// Alarm keypad FB (B11-11-11L11-11-11)
FUNCTION_BLOCK FB_AlarmKeypad IMPLEMENTS I_AlarmKeypad
VAR
	sName			: STRING;				// Keypad name

	fbButton1		: FB_DigitalIn;			// Button 1
	fbLed1			: FB_DigitalOut;		// LED 1
	fbButton2		: FB_DigitalIn;			// Button 2
	fbLed2			: FB_DigitalOut;		// LED 2
	fbButton3		: FB_DigitalIn;			// Button 3
	fbLed3			: FB_DigitalOut;		// LED 3
	fbButton4		: FB_DigitalIn;			// Button 4
	fbLed4			: FB_DigitalOut;		// LED 4
	fbButton5		: FB_DigitalIn;			// Button 5
	fbLed5			: FB_DigitalOut;		// LED 5
	fbButton6		: FB_DigitalIn;			// Button 6
	fbLed6			: FB_DigitalOut;		// LED 6
	fbBuzzer		: FB_DigitalOut;		// Buzzer

	eState			: E_KeypadState;		// Keypad state
	sConfiguredCode	: STRING;				// Configured alarm code
	sInputCode		: STRING;				// User input code
	dtInputTime		: DATE_AND_TIME;		// Date and time of last user input
	stLedsDefault	: ST_LedState;			// Default LEDs state
	
	stHMI			: ST_AlarmKeypadHMI;	// HMI data
	stVirtual		: ST_AlarmKeypadVirtual;	// Virtual keypad
END_VAR

// Returns true if the user input code equals the configured code
METHOD CheckCode : BOOL
// Compare codes
CheckCode := sInputCode = sConfiguredCode;

// Reset input if correct code was entered
IF CheckCode THEN
	Reset();
END_IF
END_METHOD

// Collect user input from buttons and build the entered code, returns true if input was detected
METHOD PRIVATE CollectInput: BOOL
VAR
	sInput			: STRING;
END_VAR
// Check buttons and translate to input
IF fbButton1.Command = E_DICommand.ShortPress THEN sInput := '1'; END_IF
IF fbButton2.Command = E_DICommand.ShortPress THEN sInput := '2'; END_IF
IF fbButton3.Command = E_DICommand.ShortPress THEN sInput := '3'; END_IF
IF fbButton4.Command = E_DICommand.ShortPress THEN sInput := '4'; END_IF
IF fbButton5.Command = E_DICommand.ShortPress THEN sInput := '5'; END_IF
IF fbButton6.Command = E_DICommand.ShortPress THEN sInput := '6'; END_IF

// Check if input was detected
IF sInput <> '' THEN
	// Build user input code
	sInputCode := CONCAT(sInputCode, sInput);
	
	// Update time of last input
	dtInputTime := GetDateTime();
	
	// Set output
	CollectInput := TRUE;
ELSE
	// Set output
	CollectInput := FALSE;
END_IF
END_METHOD

// Run this method every cycle
METHOD Execute
VAR CONSTANT
	stLedsOn	: ST_LedState := (eLed1 := E_DOCommand.On,
									eLed2 := E_DOCommand.On,
									eLed3 := E_DOCommand.On,
									eLed4 := E_DOCommand.On,
									eLed5 := E_DOCommand.On,
									eLed6 := E_DOCommand.On);
END_VAR
// Keypad state machine
CASE eState OF
	E_KeypadState.Init:
		// Initialize
		eState := E_KeypadState.Idle;
	
	E_KeypadState.Idle:
		// Wait for input
		IF CollectInput() THEN
			eState := E_KeypadState.InputDetected;
		END_IF
	
	E_KeypadState.InputDetected:
		// Collect input in every state so no input is lost
		CollectInput();
		
		// Enable all LEDs
		SetLeds(stLedsOn);
		
		eState := E_KeypadState.CheckInput;
		
	E_KeypadState.CheckInput:
		// Continue collecting input
		CollectInput();
		
		// If no input is detected during some time, reset the keypad
		IF GetDateTime() - dtInputTime > T#2S THEN
			eState := E_KeypadState.Reset;
		END_IF
		
	E_KeypadState.Reset:
		// Reset keypad
		Reset();
		
		eState := E_KeypadState.Idle;
END_CASE

// Update HMI
UpdateHMI();
END_METHOD

METHOD FB_init : BOOL
VAR_INPUT
	bInitRetains	: BOOL;		// if TRUE, the retain variables are initialized (warm start / cold start)
	bInCopyCode		: BOOL;		// if TRUE, the instance afterwards gets moved into the copy code (online change)
	
	sKeypadName		: STRING;	// Keypad name
END_VAR
sName := sKeypadName;

fbBuzzer.SetBlinkPeriod(tPeriod := T#1500MS);
END_METHOD

// Returns the HMI data
PROPERTY HmiData : ST_AlarmKeypadHMI
GET
HmiData := stHMI;
END_GET
END_PROPERTY

// Returns the keypad name
PROPERTY Name : STRING
GET
Name := sName;
END_GET
END_PROPERTY

// Reset the keypad
METHOD PRIVATE Reset
// Reset user input code
sInputCode := '';

// Reset all LEDs to their default value
SetLeds(stLedsDefault);
END_METHOD

// Call this method once when the alarm state is changed
METHOD SetAlarmState
VAR_INPUT
	eAlarmState				: E_AlarmState;		// Alarm state
END_VAR
VAR CONSTANT
	stLedsAlarmOn			: ST_LedState := (eLed1 := E_DOCommand.On,
											eLed2 := E_DOCommand.Off,
											eLed3 := E_DOCommand.Off,
											eLed4 := E_DOCommand.Off,
											eLed5 := E_DOCommand.Off,
											eLed6 := E_DOCommand.Off);
	stLedsAlarmOff			: ST_LedState := (eLed1 := E_DOCommand.Off,
											eLed2 := E_DOCommand.Off,
											eLed3 := E_DOCommand.Off,
											eLed4 := E_DOCommand.Off,
											eLed5 := E_DOCommand.Off,
											eLed6 := E_DOCommand.Off);
	stLedsAlarmEnabling		: ST_LedState := (eLed1 := E_DOCommand.Blink,
											eLed2 := E_DOCommand.Off,
											eLed3 := E_DOCommand.Off,
											eLed4 := E_DOCommand.Off,
											eLed5 := E_DOCommand.Off,
											eLed6 := E_DOCommand.Off);
	stLedsAlarmWarning		: ST_LedState := (eLed1 := E_DOCommand.Blink,
											eLed2 := E_DOCommand.Off,
											eLed3 := E_DOCommand.Off,
											eLed4 := E_DOCommand.Off,
											eLed5 := E_DOCommand.Off,
											eLed6 := E_DOCommand.Off);
	stLedsAlarmTripped		: ST_LedState := (eLed1 := E_DOCommand.Blink,
											eLed2 := E_DOCommand.Off,
											eLed3 := E_DOCommand.Off,
											eLed4 := E_DOCommand.Off,
											eLed5 := E_DOCommand.Off,
											eLed6 := E_DOCommand.Off);
	stLedsAlarmDisabling	: ST_LedState := (eLed1 := E_DOCommand.Blink,
											eLed2 := E_DOCommand.Off,
											eLed3 := E_DOCommand.Off,
											eLed4 := E_DOCommand.Off,
											eLed5 := E_DOCommand.Off,
											eLed6 := E_DOCommand.Off);
END_VAR
// Set LEDs default state
CASE eAlarmState OF
	E_AlarmState.Off:
		// Alarm is off
		stLedsDefault := stLedsAlarmOff;
		
	E_AlarmState.Enabling:
		// Alarm is enabling
		fbLed1.SetBlinkPeriod(tPeriod := T#1500MS);	// Same as buzzer
		stLedsDefault := stLedsAlarmEnabling;
	
	E_AlarmState.Enabled:
		// Alarm is on
		stLedsDefault := stLedsAlarmOn;
		
	E_AlarmState.Warning:
		// Alarm is warning
		fbLed1.SetBlinkPeriod(tPeriod := T#500MS);	// Fast blinking, buzzer is on continuously
		stLedsDefault := stLedsAlarmWarning;
		
	E_AlarmState.Tripped:
		// Alarm has been tripped
		fbLed1.SetBlinkPeriod(tPeriod := T#500MS);	// Fast blinking, alarm is sounding
		stLedsDefault := stLedsAlarmTripped;
		
	E_AlarmState.Disabling:
		// Alarm has been tripped
		fbLed1.SetBlinkPeriod(tPeriod := T#250MS);	// Fast blinking, indicate alarm is disabling
		stLedsDefault := stLedsAlarmDisabling;
END_CASE

// Reset keypad
Reset();
END_METHOD

// Set the buzzer command
METHOD SetBuzzer
VAR_INPUT
	eCommand	: E_DOCommand;
END_VAR
// Set digital output command
fbBuzzer.SetCommand(eCommandIn := eCommand);
END_METHOD

// Set the keypad configured code
METHOD SetConfiguredCode
VAR_INPUT
	sCode	:	STRING;		// Configured code
END_VAR
// Set configured alarm code
sConfiguredCode := sCode;
END_METHOD

// Set the LEDs state
METHOD PRIVATE SetLeds
VAR_INPUT
	stLeds		: ST_LedState;		// LED states
END_VAR
fbLed1.SetCommand(eCommandIn := stLeds.eLed1);
fbLed2.SetCommand(eCommandIn := stLeds.eLed2);
fbLed3.SetCommand(eCommandIn := stLeds.eLed3);
fbLed4.SetCommand(eCommandIn := stLeds.eLed4);
fbLed5.SetCommand(eCommandIn := stLeds.eLed5);
fbLed6.SetCommand(eCommandIn := stLeds.eLed6);
END_METHOD

// Update HMI
METHOD PRIVATE UpdateHMI
VAR
	stLed1HMI	: ST_HmiDigitalOut;
	stLed2HMI	: ST_HmiDigitalOut;
	stLed3HMI	: ST_HmiDigitalOut;
	stLed4HMI	: ST_HmiDigitalOut;
	stLed5HMI	: ST_HmiDigitalOut;
	stLed6HMI	: ST_HmiDigitalOut;
	stBuzzerHMI	: ST_HmiDigitalOut;
END_VAR
// Get data
stLed1HMI := fbLed1.HmiData;
stLed2HMI := fbLed2.HmiData;
stLed3HMI := fbLed3.HmiData;
stLed4HMI := fbLed4.HmiData;
stLed5HMI := fbLed5.HmiData;
stLed6HMI := fbLed6.HmiData;
stBuzzerHMI := fbBuzzer.HmiData;

// Set HMI data
stHMI.bLed1 := stLed1HMI.bValue;
stHMI.bLed2 := stLed2HMI.bValue;
stHMI.bLed3 := stLed3HMI.bValue;
stHMI.bLed4 := stLed4HMI.bValue;
stHMI.bLed5 := stLed5HMI.bValue;
stHMI.bLed6 := stLed6HMI.bValue;
stHMI.bBuzzer := stBuzzerHMI.bValue;

stHMI.sCode := sInputCode;
stHMI.sName := sName;

// Set buttons
fbButton1.SetExternalIn(bIn := stVirtual.bButton1);
fbButton2.SetExternalIn(bIn := stVirtual.bButton2);
fbButton3.SetExternalIn(bIn := stVirtual.bButton3);
fbButton4.SetExternalIn(bIn := stVirtual.bButton4);
fbButton5.SetExternalIn(bIn := stVirtual.bButton5);
fbButton6.SetExternalIn(bIn := stVirtual.bButton6);
END_METHOD

END_FUNCTION_BLOCK

(* stored: Version 1.1.0.1, ProductVersion 3.1.4024.12
   POU FB_AlarmKeypad: Id {a80355c7-d520-4b86-beb1-ae604d52844e}, SpecialFunc None
   Folder Methods: Id {ece52884-0872-4a62-a42f-6ab43354ba26}
   Folder Properties: Id {f0934509-7275-4b2a-96b4-09513f05b8dd}
   Method CheckCode: Id {3b02d97c-c990-4ebc-9bb2-3370f3699b9c}
   Method CollectInput: Id {fd4deb83-44f6-4ec5-9c14-9171b2d5e000}
   Method Execute: Id {dcfc6ac9-b1ab-4fce-abd9-3df78b1908cc}
   Method FB_init: Id {f26755b2-272a-4307-9c02-60417ea1380a}
   Property HmiData: Id {4a86c3b2-3ccf-4749-96c6-9488329c41e3}
   Get Get: Id {255b3549-d762-4caa-b1dd-4b7877205dcd}
   Property Name: Id {27c2cdd2-67b8-42bd-bda7-f79e5fc88dfd}
   Get Get: Id {9e822015-9e8f-4e75-aff4-922a47a32c24}
   Method Reset: Id {fcbf7db0-52ce-4432-89bc-348c5bf3de67}
   Method SetAlarmState: Id {8c2a4b4b-adbc-47ae-b535-c8cc81d2d62a}
   Method SetBuzzer: Id {8c85d6a6-e587-43ab-ac28-0d2066d871e3}
   Method SetConfiguredCode: Id {ea8e82ff-a600-4b6b-8104-4c28e5f58674}
   Method SetLeds: Id {4e78cd65-e66b-4185-abae-07e993abdc49}
   Method UpdateHMI: Id {7a0629e2-90c8-426c-8935-80070f3d7d43} *)
